{attribute 'qualified_only'}
VAR_GLOBAL
END_VAR

(* stored: Version 1.1.0.1, ProductVersion 3.1.4024.11
   GVL GVL_VideoPlaybackConfig: Id {21ca66e2-535e-0113-297e-0521c35af387} *)
